Universal Robots PolyScope program: IAC008 PinCount.urp

Program IAC008 PinCount (installation=default directory=/programs createdIn=5.9.1.1031110 lastSavedIn=5.9.1.1031110 robotSerialNumber=20195501059)
Calibrated DH parameters: a=[0.000146, -0.418764, -0.053981, 0.000058, -0.000023, 0]; d=[0.162545, 37.319448, -206.067439, 168.881546, 0.09955, 0.099464]; alpha=[1.57004, -0.001979, 0.002304, 1.570607, -1.57066, 0]; deltaTheta=[0, -0.174616, -1.258233, 1.432844, -0.000001, 0]
BeforeStart
  URCap Gripper Activate (Robotiq_Grippers, Robotiq Inc.) dataModel(ResetAndActivateKey=false)
  initial_p := get_actual_tcp_pose()
  MoveJ speed 60 deg/s, acceleration 80 deg/s^2 (useActiveTCP=true) feature=Base
    Waypoint Waypoint (Variable): variable=initial_p
  Set DigitalOutput pin=digital_out[1]; digitalValue=1
Robot Program (runOnlyOnce=false)
  URCap Gripper (Robotiq_Grippers, Robotiq Inc.) dataModel(position=100.0, force=100.0, speed=100.0, positionInDouble=100.0, forceInDouble=100.0, speedInDouble=100.0, slaveIds=[9], blocking=true)
  MoveL speed 250 mm/s, acceleration 1200 mm/s^2 (useActiveTCP=true) feature=Base
    Waypoint home: TCP in base x=353.442 y=-425.051 z=15.364 mm, rx=-2.1827 ry=-2.2594 rz=0 rad; joints [115.734, -68.978, 112.532, -133.544, 270.037, 113.795] deg; TCP offset x=0 y=0 z=174 mm, rx=0 ry=0 rz=0 rad
  Call vision_connect
  MoveL speed 250 mm/s, acceleration 1200 mm/s^2 (useActiveTCP=true) feature=Base
    Waypoint inspect: TCP in base x=195.186 y=-428.085 z=202.343 mm, rx=1.174 ry=2.7663 rz=-0.4003 rad; joints [99.729, -101.18, 122.479, -127.473, 267.218, 55.335] deg
  Loop Counting (count=10) loopVariable(name=Loop_3)
    MoveL speed 250 mm/s, acceleration 1200 mm/s^2 (useActiveTCP=true) feature=Base
      Call vision_pincount
      If nPins≠16
        Popup Error (haltProgram=false message=Did not find 16 pins inputType=Text)
      MoveDirectionNode (toolParams=0.25, 0.5) expression=[-1.0,-1.0,0.0]; feature=Base
        Until DISTANCE (allowActions=false deceleration=3 distanceNodeType=STOP) Distance=0.001; motionParameters(blendRadius=0)
  MoveL speed 250 mm/s, acceleration 1200 mm/s^2 (useActiveTCP=true) feature=Base
    Waypoint home: TCP in base x=353.442 y=-425.051 z=15.364 mm, rx=-2.1827 ry=-2.2594 rz=0 rad; joints [115.734, -68.978, 112.532, -133.544, 270.037, 113.795] deg
  Call vision_disconnect
SubProgram  [hidden by the author, left out]
SubProgram  [hidden by the author, left out]
SubProgram  [hidden by the author, left out]
SubProgram vision_connect [hidden by the author, left out]
SubProgram vision_pincount [hidden by the author, left out]
SubProgram vision_disconnect [hidden by the author, left out]
